(* Logix 5000 project; controller cal1615 1756-L62 rev 20.11; software revision 20.05; part 9 of 82 *)
(* tags used below, declared in another part *)
   FAULT : BOOL;   // Fault AFI
   p01_ai_prs : REAL;   // System Inputs Oxidizer Differential Pressure
   p01_ai_tc : REAL;   // System Inputs Oxidizer Inlet Temperature
   p01_di_edge_ctrl_estop_active : BOOL;   // System Digital Input Edge Control Estop Active
   p01_di_estop_1_tripped : BOOL;   // System Digital Input EStop Relay 1 Tripped
   p01_di_estop_2_tripped : BOOL;   // System Digital Input EStop Relay 2 Tripped
   p01_di_estop_reset : BOOL;   // System Digital Inupt Main Operator Panel E-Stop Reset
   p01_di_impreg_estop_active : BOOL;   // System Digital Input Impreg Estop Active
   p01_di_letoff_estop_active : BOOL;   // System Digital Input Letoff Estop Active
   p01_di_lof_acc_estop_active : BOOL;   // System Digital Input Letoff Accumulator Estop Active
   p01_di_main_hmi_estop : BOOL;   // System Digital Inupt Main Operator Panel E-Stop Active
   p01_di_rope_sw_1_active : BOOL;   // System Digital Input Rope Switch 1 Active
   p01_di_rope_sw_2_active : BOOL;   // System Digital Input Rope Switch 2 Active
   p01_di_rope_sw_3_active : BOOL;   // System Digital Input Rope Switch 3 Active
   p01_di_rope_sw_4_active : BOOL;   // System Digital Input Rope Switch 4 Active
   p01_di_rope_sw_5_active : BOOL;   // System Digital Input Rope Switch 5 Active
   p01_di_rope_sw_6_active : BOOL;   // System Digital Input Rope Switch 6 Active
   p01_di_rope_sw_7_active : BOOL;   // System Digital Input Rope Switch 7 Active
   p01_di_rope_sw_8_active : BOOL;   // System Digital Input Rope Switch 8 Active
   p01_di_splice_estop_active : BOOL;   // System Digital Input Splice Press Estop Active
   p01_di_ts2_estop_active : BOOL;   // System Digital Input Tension Stand 2 Estop Active
   p01_di_winder_estop_active : BOOL;   // System Digital Input Winder Estop Active
   p01_dint_to_hmi : DINT[16];   // System Dint to HMI
   p01_int_from_oxidizer : INT[10];   // System Oxidizer Int from Oxidizer
   p01r01 : routine;
   p01r02 : routine;   // System Misc Control
   p01r02_all_fans_stopped : BOOL;   // System Misc Control All Fans Stopped
   p01r02_batch_run_time_hrs : DINT;   // System Misc Control Batch Hours
   p01r02_do_horn : BOOL;   // System Outputs Horn
   p01r02_ethernet_comm : DINT;
   p01r02_horn : BOOL;
   p01r02_plc_faults : DINT;   // System Misc Control PLC Faults
   p01r02_timer_fault : TIMER[25];   // System Misc Control Fault Dwell Timer
   p01r02_timer_half_second_on : TIMER;   // System Misc Control Timer 1/2 Second Pulse On
   p01r02_timer_second : TIMER[2];   // System Misc Control Timer Second Pulse
   p01r02_timer_warning : TIMER[4];   // System Misc Control Warning Delay
   p01r03 : routine;   // System Inputs
   p01r03_oxidizer_prs : SYS_SCP;   // System Inputs Oxidizer Differential Pressure Scaling
   p01r03_prs_input_max : REAL;
   p01r03_prs_input_min : REAL;
   p01r03_prs_output_max : REAL;
   p01r03_prs_output_min : REAL;
   p01r03_timer_fault : TIMER[4];   // System Input Fault Delay
   p01r03_timer_warning : TIMER[4];   // System Input Warning Delay
   p01r04 : routine;   // System Outputs
   p01r04_LFL_warning : BOOL;   // System Misc Control LFL Warning
   p01r04_Temp_deviation_warning : BOOL;   // System Misc Control Temperature Deviation Warning
   p01r04_timer_fault : TIMER[4];   // System Output Fault Delay
   p01r04_timer_warning : TIMER[4];   // System Output Warning Delay
   p01r05 : routine;   // System Dint to HMI
   p01r05_enc : SYS_ENC;   // System Dint to HMI Encoder
   p01r05_timer_fault : TIMER[4];   // System Dint to HMI Fault Delay
   p01r09_mode_jog : BOOL;   // System Modes Jog Mode
   p01r09_mode_run : BOOL;   // System Modes All Modes Run Mode
   p01r09_mode_thread : BOOL;   // System Modes Thread Mode
   p01r09_open_oven : BOOL;
   p01r09_pb_global_reset : BOOL;   // System Modes PB: Global Fault Reset
   p01r10_fault_exists : BOOL;
   p01r10_unack_fault_ex : BOOL;
   p01r10_unack_warn_ex : BOOL;   // System Annunciators Unacknowledged Warning Exists
   p01r10_warning_exists : BOOL;
   p01r13_line_running : BOOL;   // System Line Start Sequence Line Running
   p01r13_status : DINT;   // System Line Start Sequence Encoded Step
   p01r14_oxidizer_heart_beat_ok : BOOL;   // System Oxidizer Heart Beat Ok
   p11r12_Oven_auto_run_on : BOOL;   // Zone 1 Temp Sequence Oven Auto Run On
(* P01_System, continued *)

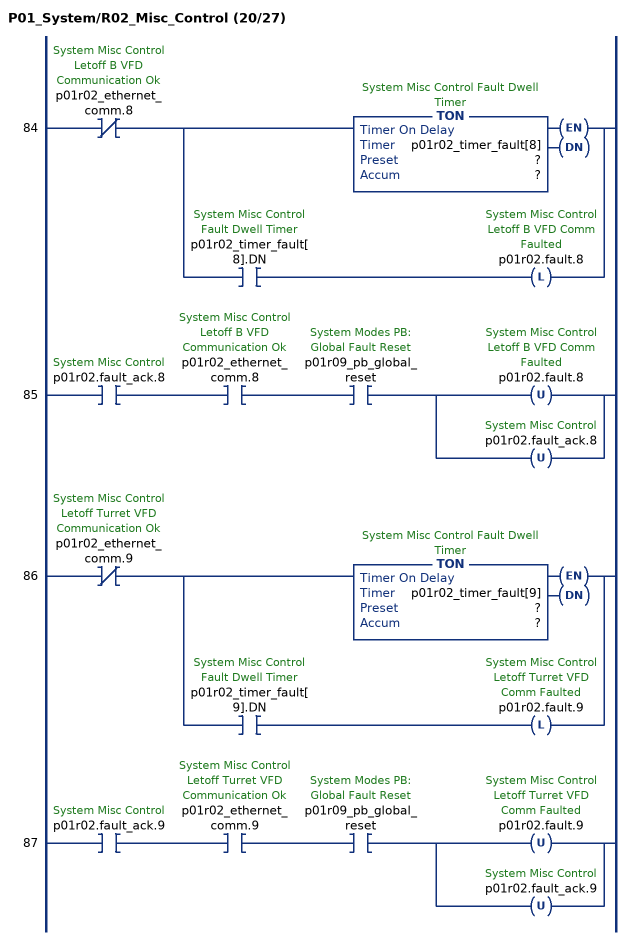
   [picture p67: P01_System/R02_Misc_Control rungs 84-87]
   84: XIO(p01r02_ethernet_comm.8)[TON(p01r02_timer_fault[8],?,?) ,XIC(p01r02_timer_fault[8].DN) OTL(p01r02.fault.8) ];
   85: XIC(p01r02.fault_ack.8)XIC(p01r02_ethernet_comm.8)XIC(p01r09_pb_global_reset)[OTU(p01r02.fault.8) ,OTU(p01r02.fault_ack.8) ];
   86: XIO(p01r02_ethernet_comm.9)[TON(p01r02_timer_fault[9],?,?) ,XIC(p01r02_timer_fault[9].DN) OTL(p01r02.fault.9) ];
   87: XIC(p01r02.fault_ack.9)XIC(p01r02_ethernet_comm.9)XIC(p01r09_pb_global_reset)[OTU(p01r02.fault.9) ,OTU(p01r02.fault_ack.9) ];
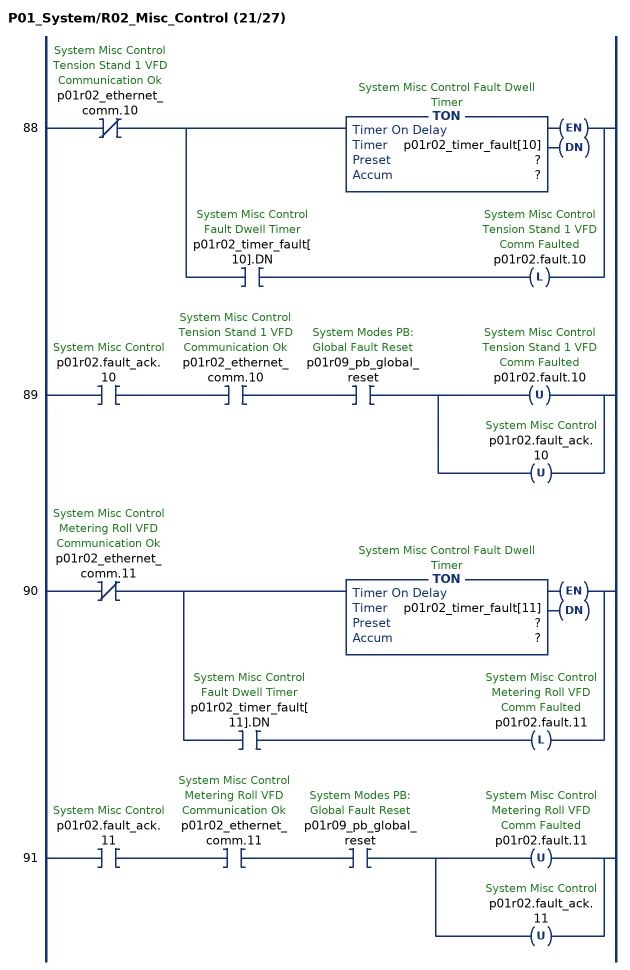
   88: XIO(p01r02_ethernet_comm.10)[TON(p01r02_timer_fault[10],?,?) ,XIC(p01r02_timer_fault[10].DN) OTL(p01r02.fault.10) ];
   89: XIC(p01r02.fault_ack.10)XIC(p01r02_ethernet_comm.10)XIC(p01r09_pb_global_reset)[OTU(p01r02.fault.10) ,OTU(p01r02.fault_ack.10) ];
   90: XIO(p01r02_ethernet_comm.11)[TON(p01r02_timer_fault[11],?,?) ,XIC(p01r02_timer_fault[11].DN) OTL(p01r02.fault.11) ];
   91: XIC(p01r02.fault_ack.11)XIC(p01r02_ethernet_comm.11)XIC(p01r09_pb_global_reset)[OTU(p01r02.fault.11) ,OTU(p01r02.fault_ack.11) ];
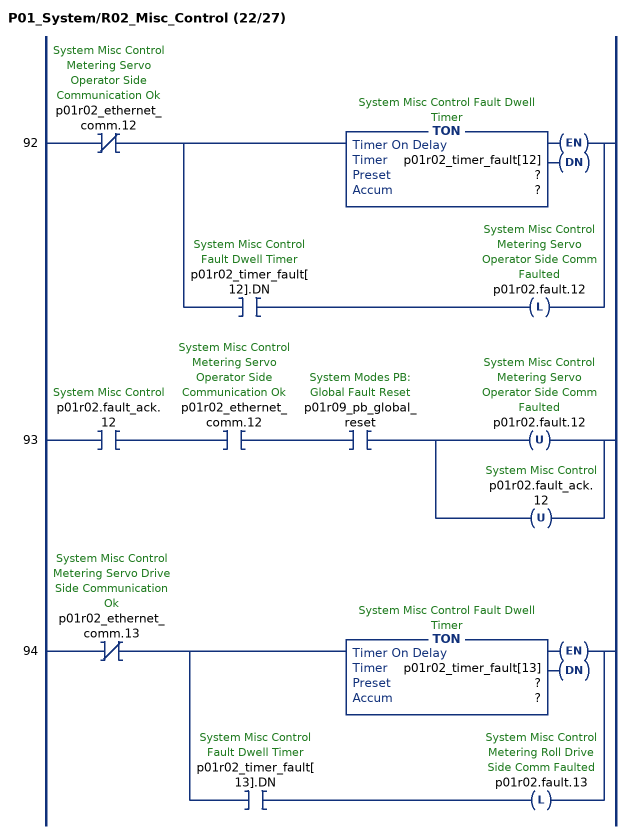
   92: XIO(p01r02_ethernet_comm.12)[TON(p01r02_timer_fault[12],?,?) ,XIC(p01r02_timer_fault[12].DN) OTL(p01r02.fault.12) ];
   93: XIC(p01r02.fault_ack.12)XIC(p01r02_ethernet_comm.12)XIC(p01r09_pb_global_reset)[OTU(p01r02.fault.12) ,OTU(p01r02.fault_ack.12) ];
   94: XIO(p01r02_ethernet_comm.13)[TON(p01r02_timer_fault[13],?,?) ,XIC(p01r02_timer_fault[13].DN) OTL(p01r02.fault.13) ];
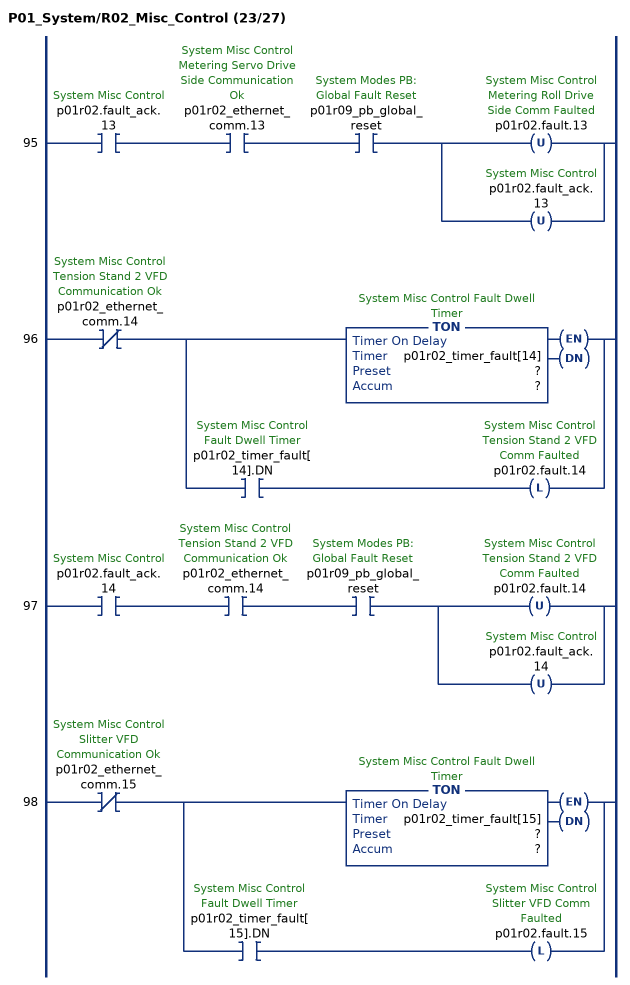
   95: XIC(p01r02.fault_ack.13)XIC(p01r02_ethernet_comm.13)XIC(p01r09_pb_global_reset)[OTU(p01r02.fault.13) ,OTU(p01r02.fault_ack.13) ];
   96: XIO(p01r02_ethernet_comm.14)[TON(p01r02_timer_fault[14],?,?) ,XIC(p01r02_timer_fault[14].DN) OTL(p01r02.fault.14) ];
   97: XIC(p01r02.fault_ack.14)XIC(p01r02_ethernet_comm.14)XIC(p01r09_pb_global_reset)[OTU(p01r02.fault.14) ,OTU(p01r02.fault_ack.14) ];
   98: XIO(p01r02_ethernet_comm.15)[TON(p01r02_timer_fault[15],?,?) ,XIC(p01r02_timer_fault[15].DN) OTL(p01r02.fault.15) ];
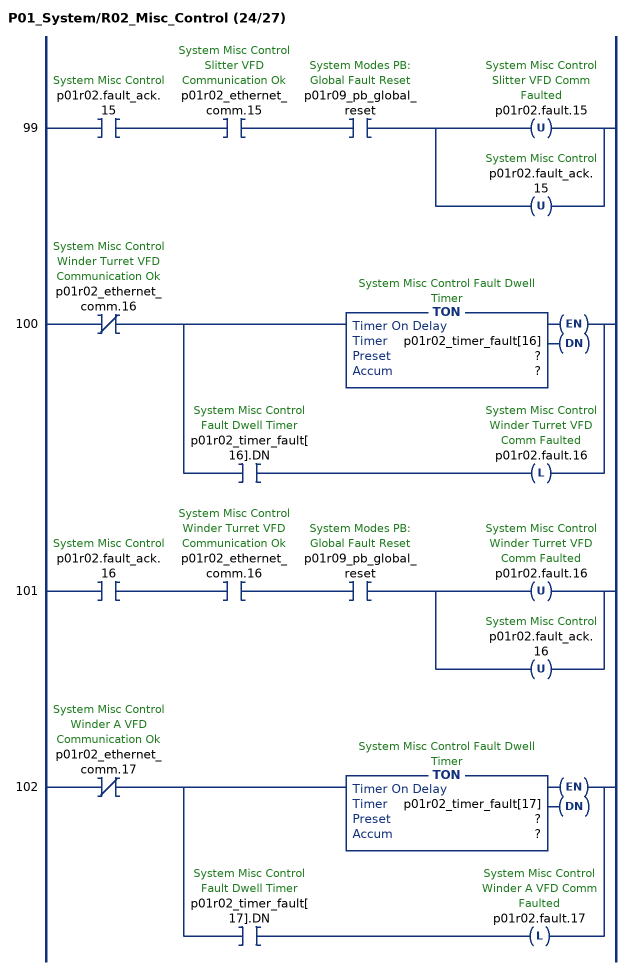
   99: XIC(p01r02.fault_ack.15)XIC(p01r02_ethernet_comm.15)XIC(p01r09_pb_global_reset)[OTU(p01r02.fault.15) ,OTU(p01r02.fault_ack.15) ];
   100: XIO(p01r02_ethernet_comm.16)[TON(p01r02_timer_fault[16],?,?) ,XIC(p01r02_timer_fault[16].DN) OTL(p01r02.fault.16) ];
   101: XIC(p01r02.fault_ack.16)XIC(p01r02_ethernet_comm.16)XIC(p01r09_pb_global_reset)[OTU(p01r02.fault.16) ,OTU(p01r02.fault_ack.16) ];
   102: XIO(p01r02_ethernet_comm.17)[TON(p01r02_timer_fault[17],?,?) ,XIC(p01r02_timer_fault[17].DN) OTL(p01r02.fault.17) ];
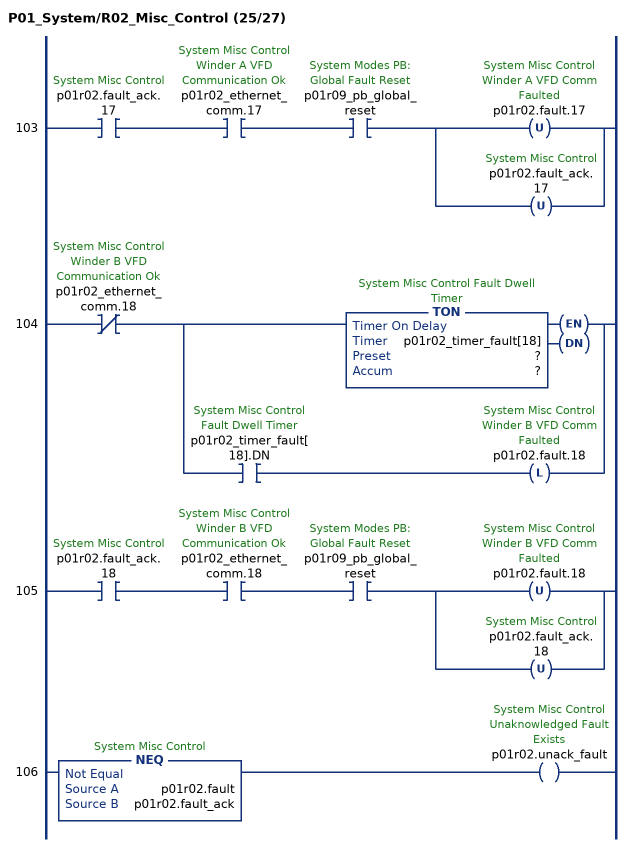
   103: XIC(p01r02.fault_ack.17)XIC(p01r02_ethernet_comm.17)XIC(p01r09_pb_global_reset)[OTU(p01r02.fault.17) ,OTU(p01r02.fault_ack.17) ];
   104: XIO(p01r02_ethernet_comm.18)[TON(p01r02_timer_fault[18],?,?) ,XIC(p01r02_timer_fault[18].DN) OTL(p01r02.fault.18) ];
   105: XIC(p01r02.fault_ack.18)XIC(p01r02_ethernet_comm.18)XIC(p01r09_pb_global_reset)[OTU(p01r02.fault.18) ,OTU(p01r02.fault_ack.18) ];
   106: NEQ(p01r02.fault,p01r02.fault_ack)OTE(p01r02.unack_fault);
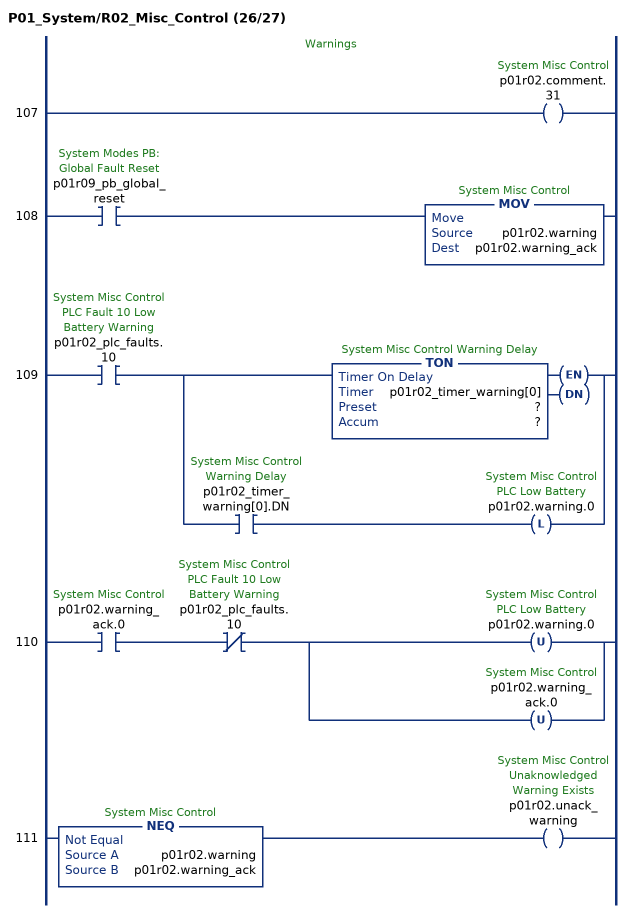
   // Warnings
   107: OTE(p01r02.comment.31);
   108: XIC(p01r09_pb_global_reset)MOV(p01r02.warning,p01r02.warning_ack);
   109: XIC(p01r02_plc_faults.10)[TON(p01r02_timer_warning[0],?,?) ,XIC(p01r02_timer_warning[0].DN) OTL(p01r02.warning.0) ];
   110: XIC(p01r02.warning_ack.0)XIO(p01r02_plc_faults.10)[OTU(p01r02.warning.0) ,OTU(p01r02.warning_ack.0) ];
   111: NEQ(p01r02.warning,p01r02.warning_ack)OTE(p01r02.unack_warning);
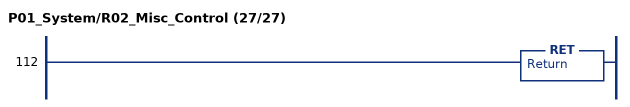
   112: RET();
END_ROUTINE

ROUTINE R03_Inputs   (* ladder *)
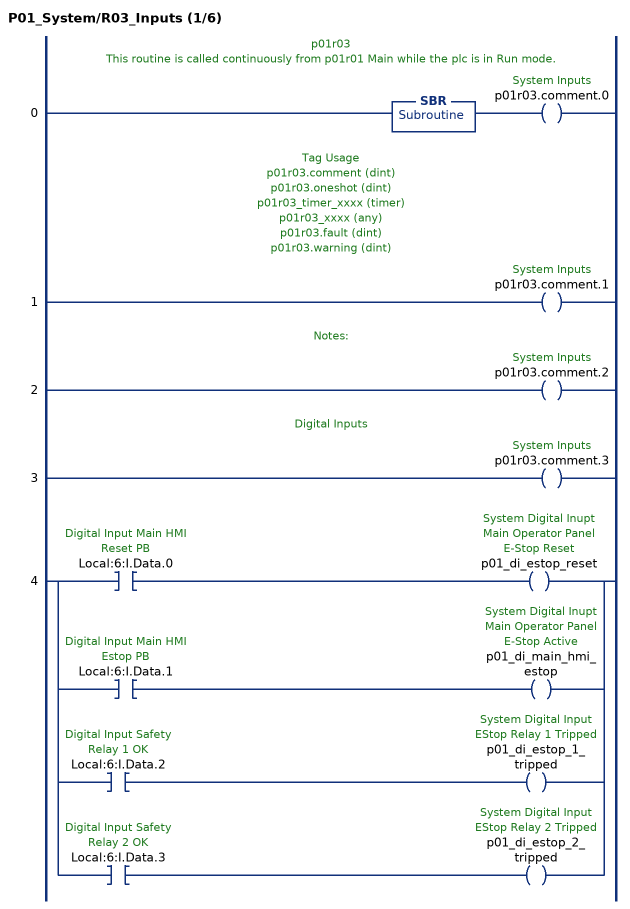
   // p01r03
   // This routine is called continuously from p01r01 Main while the plc is in Run mode.
   0: SBR()OTE(p01r03.comment.0);
   // Tag Usage
   // p01r03.comment (dint)
   // p01r03.oneshot (dint)
   // p01r03_timer_xxxx (timer)
   // p01r03_xxxx (any)
   // p01r03.fault (dint)
   // p01r03.warning (dint)
   1: OTE(p01r03.comment.1);
   // Notes:
   2: OTE(p01r03.comment.2);
   // Digital Inputs
   3: OTE(p01r03.comment.3);
   4: [XIC(Local:6:I.Data.0) OTE(p01_di_estop_reset) ,XIC(Local:6:I.Data.1) OTE(p01_di_main_hmi_estop) ,XIC(Local:6:I.Data.2) OTE(p01_di_estop_1_tripped) ,XIC(Local:6:I.Data.3) OTE(p01_di_estop_2_tripped) ];
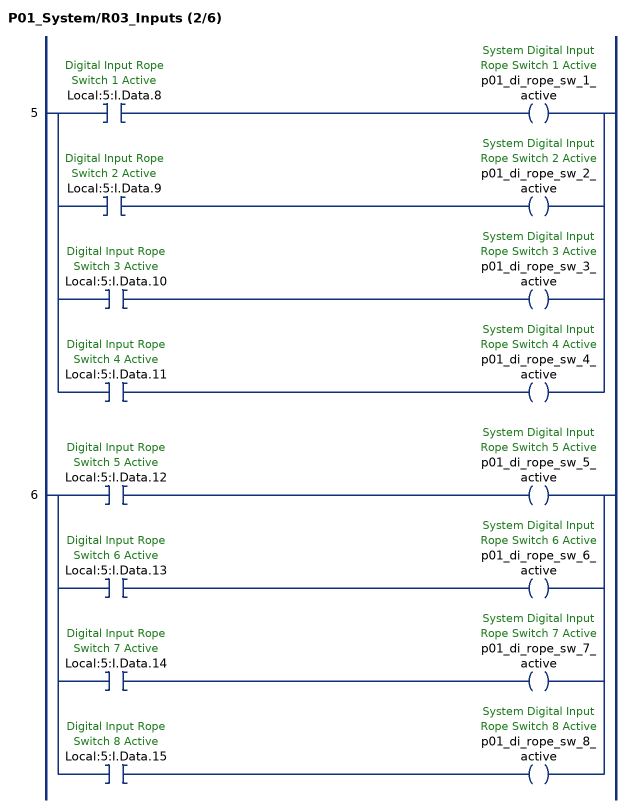
   5: [XIC(Local:5:I.Data.8) OTE(p01_di_rope_sw_1_active) ,XIC(Local:5:I.Data.9) OTE(p01_di_rope_sw_2_active) ,XIC(Local:5:I.Data.10) OTE(p01_di_rope_sw_3_active) ,XIC(Local:5:I.Data.11) OTE(p01_di_rope_sw_4_active) ];
   6: [XIC(Local:5:I.Data.12) OTE(p01_di_rope_sw_5_active) ,XIC(Local:5:I.Data.13) OTE(p01_di_rope_sw_6_active) ,XIC(Local:5:I.Data.14) OTE(p01_di_rope_sw_7_active) ,XIC(Local:5:I.Data.15) OTE(p01_di_rope_sw_8_active) ];
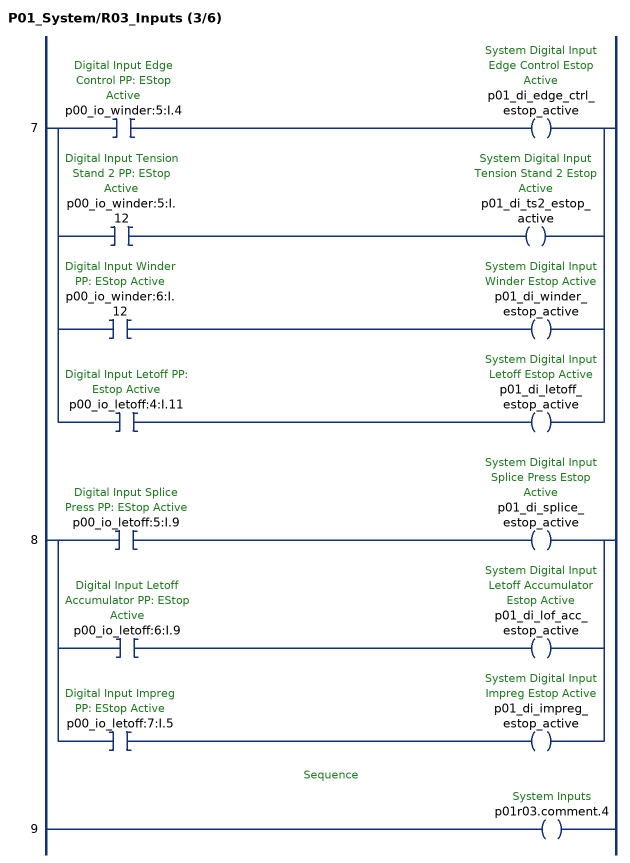
   7: [XIC(p00_io_winder:5:I.4) OTE(p01_di_edge_ctrl_estop_active) ,XIC(p00_io_winder:5:I.12) OTE(p01_di_ts2_estop_active) ,XIC(p00_io_winder:6:I.12) OTE(p01_di_winder_estop_active) ,XIC(p00_io_letoff:4:I.11) OTE(p01_di_letoff_estop_active) ];
   8: [XIC(p00_io_letoff:5:I.9) OTE(p01_di_splice_estop_active) ,XIC(p00_io_letoff:6:I.9) OTE(p01_di_lof_acc_estop_active) ,XIC(p00_io_letoff:7:I.5) OTE(p01_di_impreg_estop_active) ];
   // Sequence
   9: OTE(p01r03.comment.4);
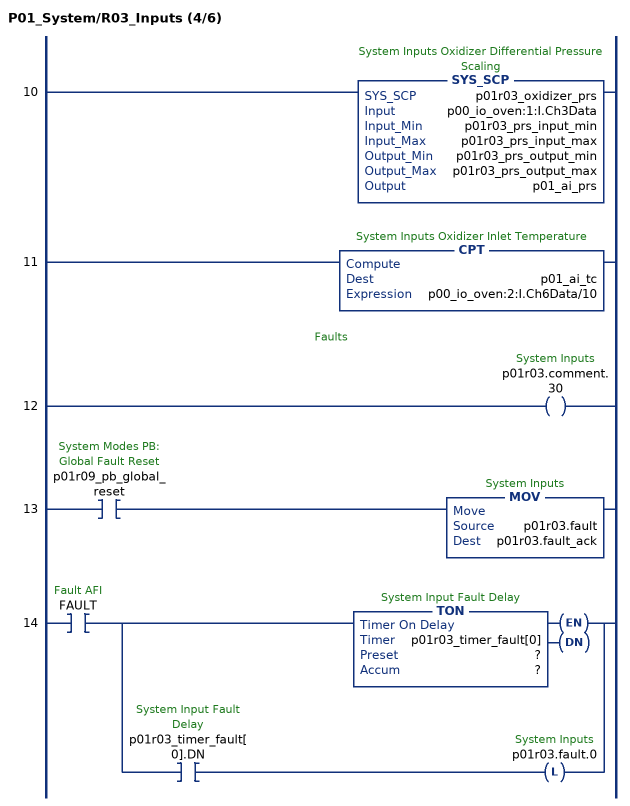
   10: SYS_SCP(p01r03_oxidizer_prs,p00_io_oven:1:I.Ch3Data,p01r03_prs_input_min,p01r03_prs_input_max,p01r03_prs_output_min,p01r03_prs_output_max,p01_ai_prs);
   11: CPT(p01_ai_tc,p00_io_oven:2:I.Ch6Data/10);
   // Faults
   12: OTE(p01r03.comment.30);
   13: XIC(p01r09_pb_global_reset)MOV(p01r03.fault,p01r03.fault_ack);
   14: XIC(FAULT)[TON(p01r03_timer_fault[0],?,?) ,XIC(p01r03_timer_fault[0].DN) OTL(p01r03.fault.0) ];
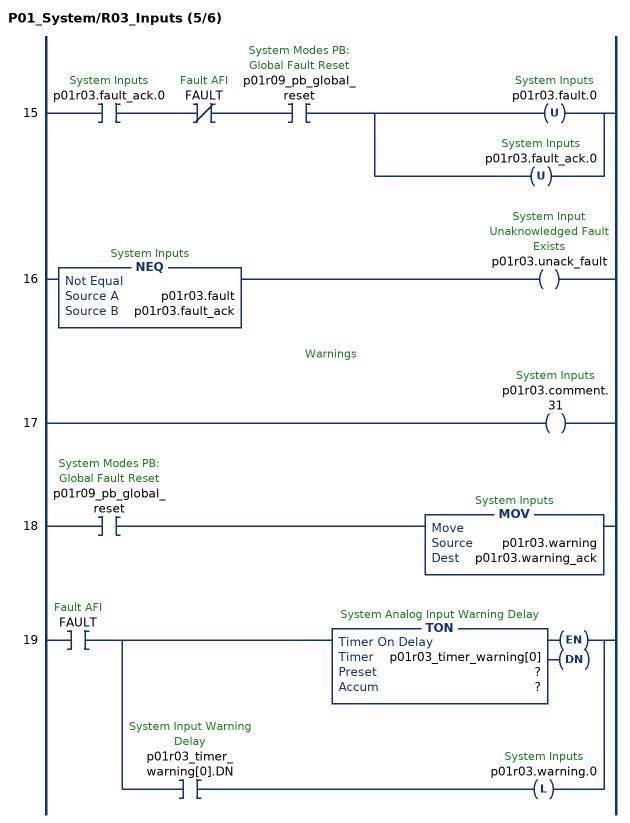
   15: XIC(p01r03.fault_ack.0)XIO(FAULT)XIC(p01r09_pb_global_reset)[OTU(p01r03.fault.0) ,OTU(p01r03.fault_ack.0) ];
   16: NEQ(p01r03.fault,p01r03.fault_ack)OTE(p01r03.unack_fault);
   // Warnings
   17: OTE(p01r03.comment.31);
   18: XIC(p01r09_pb_global_reset)MOV(p01r03.warning,p01r03.warning_ack);
   19: XIC(FAULT)[TON(p01r03_timer_warning[0],?,?) ,XIC(p01r03_timer_warning[0].DN) OTL(p01r03.warning.0) ];
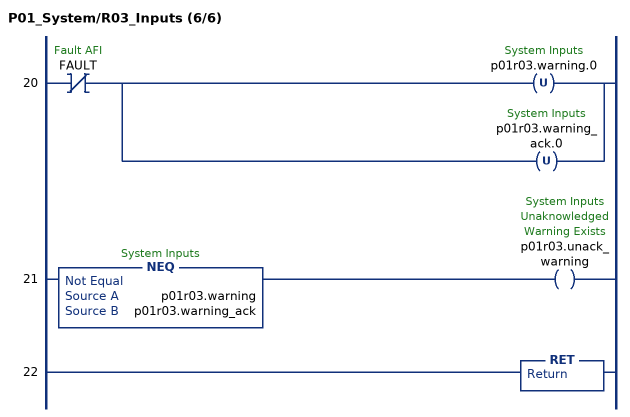
   20: XIO(FAULT)[OTU(p01r03.warning.0) ,OTU(p01r03.warning_ack.0) ];
   21: NEQ(p01r03.warning,p01r03.warning_ack)OTE(p01r03.unack_warning);
   22: RET();
END_ROUTINE

ROUTINE R04_Outputs   (* ladder *)
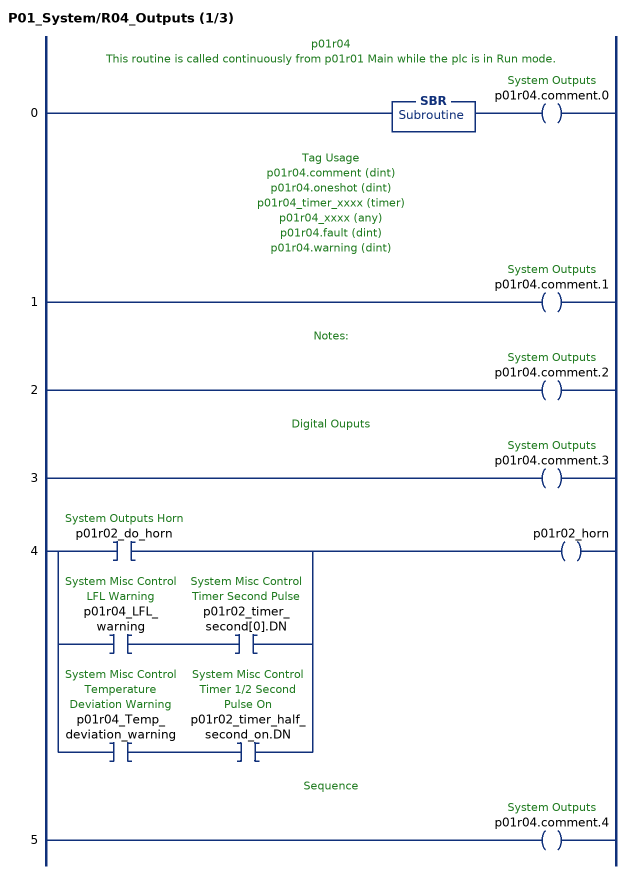
   // p01r04
   // This routine is called continuously from p01r01 Main while the plc is in Run mode.
   0: SBR()OTE(p01r04.comment.0);
   // Tag Usage
   // p01r04.comment (dint)
   // p01r04.oneshot (dint)
   // p01r04_timer_xxxx (timer)
   // p01r04_xxxx (any)
   // p01r04.fault (dint)
   // p01r04.warning (dint)
   1: OTE(p01r04.comment.1);
   // Notes:
   2: OTE(p01r04.comment.2);
   // Digital Ouputs
   3: OTE(p01r04.comment.3);
   4: [XIC(p01r02_do_horn) ,XIC(p01r04_LFL_warning) XIC(p01r02_timer_second[0].DN) ,XIC(p01r04_Temp_deviation_warning) XIC(p01r02_timer_half_second_on.DN) ]OTE(p01r02_horn);
   // Sequence
   5: OTE(p01r04.comment.4);
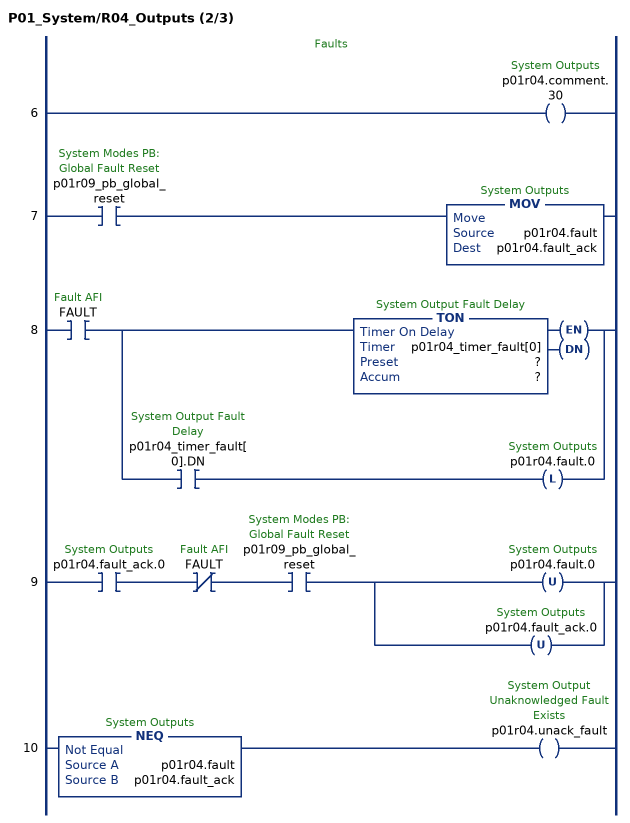
   // Faults
   6: OTE(p01r04.comment.30);
   7: XIC(p01r09_pb_global_reset)MOV(p01r04.fault,p01r04.fault_ack);
   8: XIC(FAULT)[TON(p01r04_timer_fault[0],?,?) ,XIC(p01r04_timer_fault[0].DN) OTL(p01r04.fault.0) ];
   9: XIC(p01r04.fault_ack.0)XIO(FAULT)XIC(p01r09_pb_global_reset)[OTU(p01r04.fault.0) ,OTU(p01r04.fault_ack.0) ];
   10: NEQ(p01r04.fault,p01r04.fault_ack)OTE(p01r04.unack_fault);
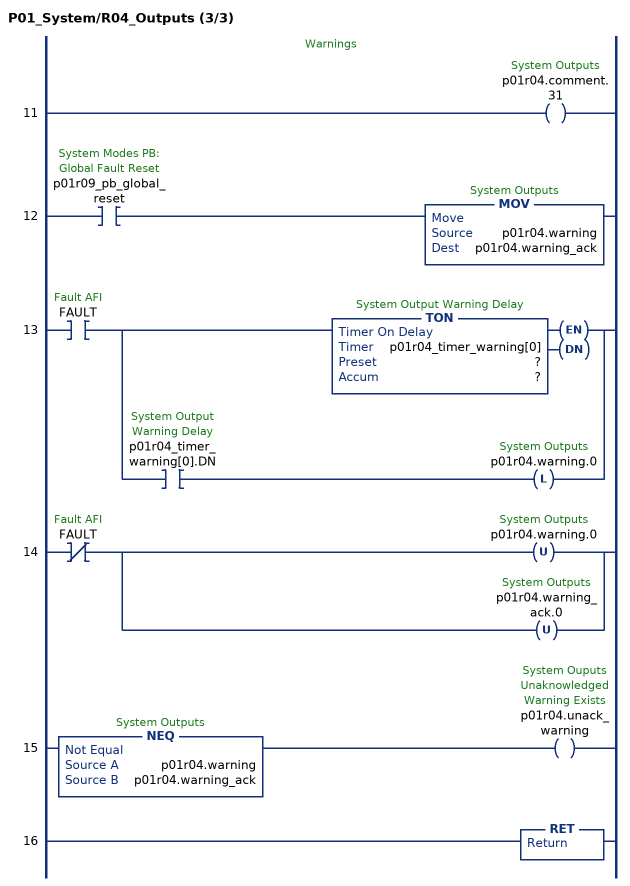
   // Warnings
   11: OTE(p01r04.comment.31);
   12: XIC(p01r09_pb_global_reset)MOV(p01r04.warning,p01r04.warning_ack);
   13: XIC(FAULT)[TON(p01r04_timer_warning[0],?,?) ,XIC(p01r04_timer_warning[0].DN) OTL(p01r04.warning.0) ];
   14: XIO(FAULT)[OTU(p01r04.warning.0) ,OTU(p01r04.warning_ack.0) ];
   15: NEQ(p01r04.warning,p01r04.warning_ack)OTE(p01r04.unack_warning);
   16: RET();
END_ROUTINE

ROUTINE R05_Dint_to_HMI   (* ladder *)
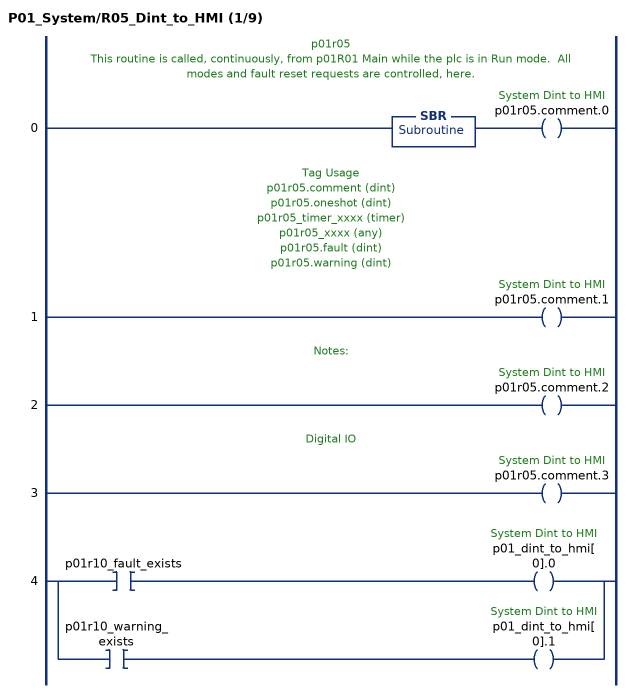
   // p01r05
   // This routine is called, continuously, from p01R01 Main while the plc is in Run mode.  All modes and fault reset requests are controlled, here.
   0: SBR()OTE(p01r05.comment.0);
   // Tag Usage
   // p01r05.comment (dint)
   // p01r05.oneshot (dint)
   // p01r05_timer_xxxx (timer)
   // p01r05_xxxx (any)
   // p01r05.fault (dint)
   // p01r05.warning (dint)
   1: OTE(p01r05.comment.1);
   // Notes:
   2: OTE(p01r05.comment.2);
   // Digital IO
   3: OTE(p01r05.comment.3);
   4: [XIC(p01r10_fault_exists) OTE(p01_dint_to_hmi[0].0) ,XIC(p01r10_warning_exists) OTE(p01_dint_to_hmi[0].1) ];
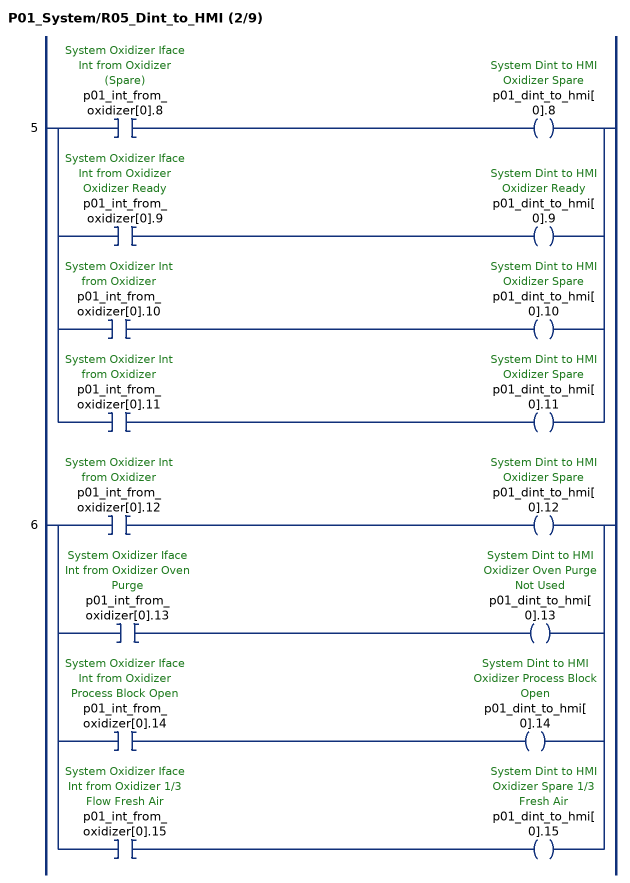
   5: [XIC(p01_int_from_oxidizer[0].8) OTE(p01_dint_to_hmi[0].8) ,XIC(p01_int_from_oxidizer[0].9) OTE(p01_dint_to_hmi[0].9) ,XIC(p01_int_from_oxidizer[0].10) OTE(p01_dint_to_hmi[0].10) ,XIC(p01_int_from_oxidizer[0].11) OTE(p01_dint_to_hmi[0].11) ];
   6: [XIC(p01_int_from_oxidizer[0].12) OTE(p01_dint_to_hmi[0].12) ,XIC(p01_int_from_oxidizer[0].13) OTE(p01_dint_to_hmi[0].13) ,XIC(p01_int_from_oxidizer[0].14) OTE(p01_dint_to_hmi[0].14) ,XIC(p01_int_from_oxidizer[0].15) OTE(p01_dint_to_hmi[0].15) ];
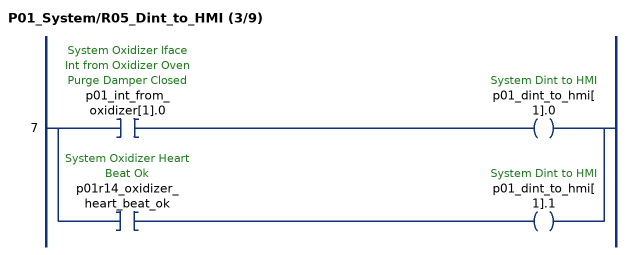
   7: [XIC(p01_int_from_oxidizer[1].0) OTE(p01_dint_to_hmi[1].0) ,XIC(p01r14_oxidizer_heart_beat_ok) OTE(p01_dint_to_hmi[1].1) ];
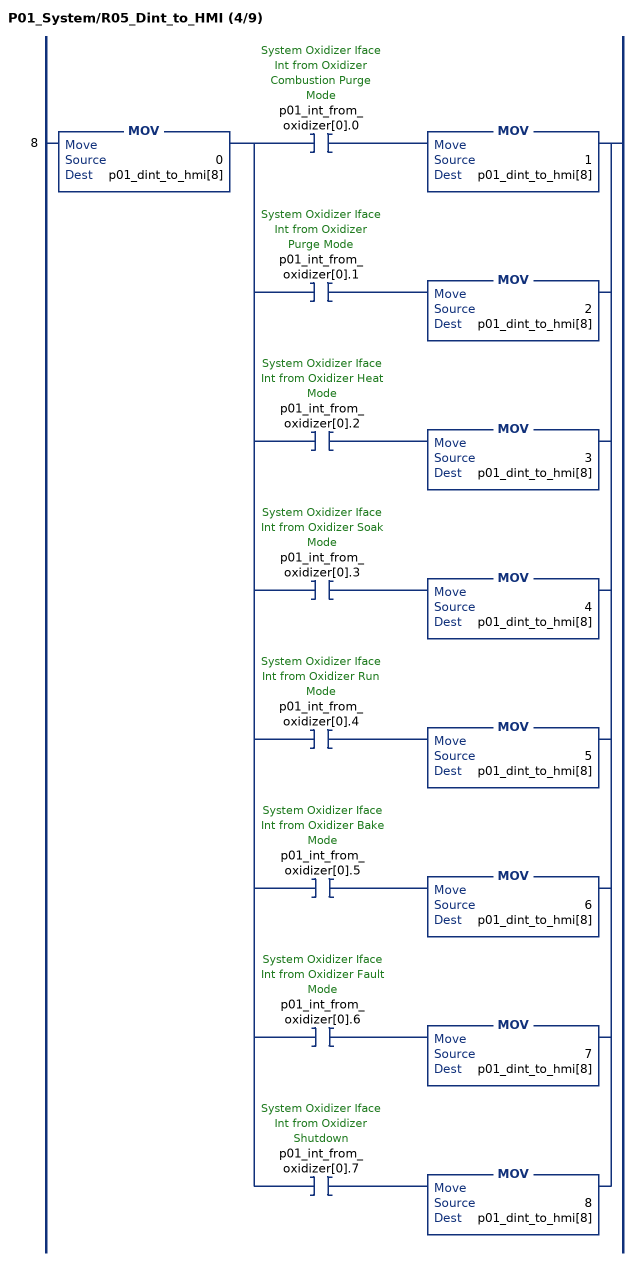
   8: MOV(0,p01_dint_to_hmi[8])[XIC(p01_int_from_oxidizer[0].0) MOV(1,p01_dint_to_hmi[8]) ,XIC(p01_int_from_oxidizer[0].1) MOV(2,p01_dint_to_hmi[8]) ,XIC(p01_int_from_oxidizer[0].2) MOV(3,p01_dint_to_hmi[8]) ,XIC(p01_int_from_oxidizer[0].3) MOV(4,p01_dint_to_hmi[8]) ,XIC(p01_int_from_oxidizer[0].4) MOV(5,p01_dint_to_hmi[8]) ,XIC(p01_int_from_oxidizer[0].5) MOV(6,p01_dint_to_hmi[8]) ,XIC(p01_int_from_oxidizer[0].6) MOV(7,p01_dint_to_hmi[8]) ,XIC(p01_int_from_oxidizer[0].7) MOV(8,p01_dint_to_hmi[8]) ];
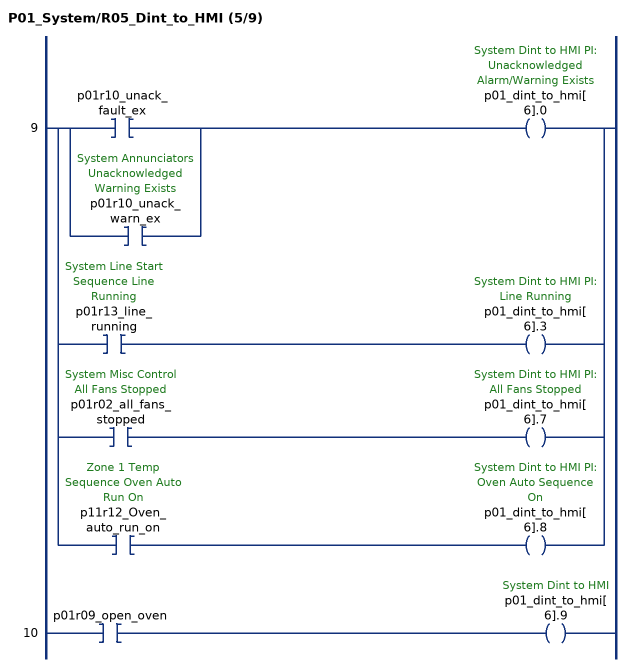
   9: [[XIC(p01r10_unack_fault_ex) ,XIC(p01r10_unack_warn_ex) ] OTE(p01_dint_to_hmi[6].0) ,XIC(p01r13_line_running) OTE(p01_dint_to_hmi[6].3) ,XIC(p01r02_all_fans_stopped) OTE(p01_dint_to_hmi[6].7) ,XIC(p11r12_Oven_auto_run_on) OTE(p01_dint_to_hmi[6].8) ];
   10: XIC(p01r09_open_oven)OTE(p01_dint_to_hmi[6].9);
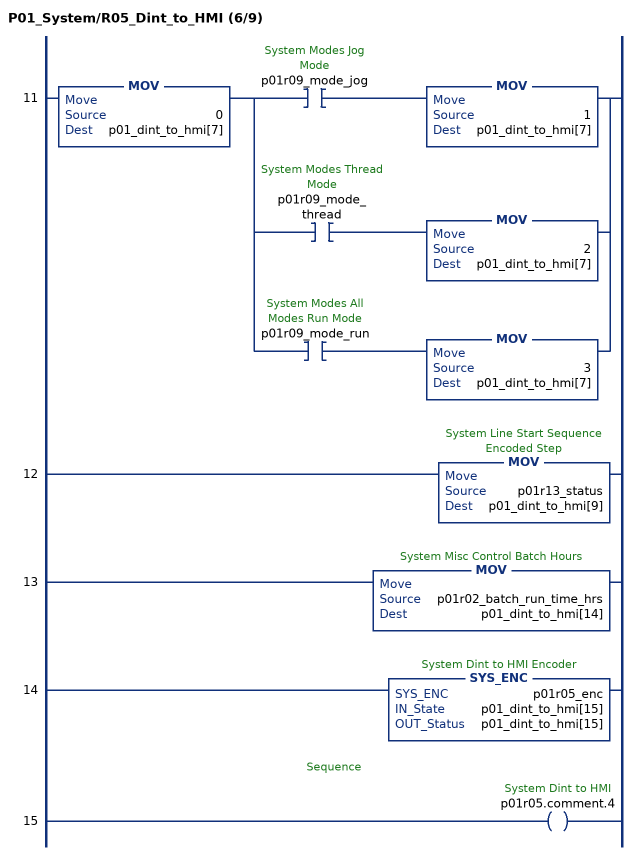
   11: MOV(0,p01_dint_to_hmi[7])[XIC(p01r09_mode_jog) MOV(1,p01_dint_to_hmi[7]) ,XIC(p01r09_mode_thread) MOV(2,p01_dint_to_hmi[7]) ,XIC(p01r09_mode_run) MOV(3,p01_dint_to_hmi[7]) ];
   12: MOV(p01r13_status,p01_dint_to_hmi[9]);
   13: MOV(p01r02_batch_run_time_hrs,p01_dint_to_hmi[14]);
   14: SYS_ENC(p01r05_enc,p01_dint_to_hmi[15],p01_dint_to_hmi[15]);
   // Sequence
   15: OTE(p01r05.comment.4);
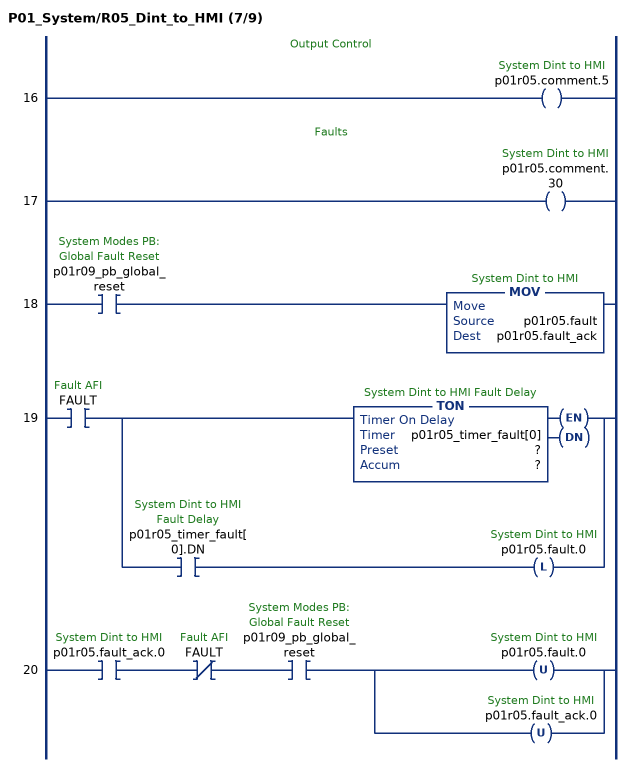
   // Output Control
   16: OTE(p01r05.comment.5);
   // Faults
   17: OTE(p01r05.comment.30);
   18: XIC(p01r09_pb_global_reset)MOV(p01r05.fault,p01r05.fault_ack);
   19: XIC(FAULT)[TON(p01r05_timer_fault[0],?,?) ,XIC(p01r05_timer_fault[0].DN) OTL(p01r05.fault.0) ];
   20: XIC(p01r05.fault_ack.0)XIO(FAULT)XIC(p01r09_pb_global_reset)[OTU(p01r05.fault.0) ,OTU(p01r05.fault_ack.0) ];
